(* Schneider Machine Expert - Basic project Questao3.3_FelipeV1_20241008, file version 2.9.0.0 *)
(* ProjectInformations: Name=Novo projeto *)

HARDWARE
  Cpu 0: TM221M16R/G
  EthernetConfiguration: NetworkName=M221, IpAllocationMode=FixedAddress, IpAddress=0.0.0.0, SubnetMask=0.0.0.0
  SerialLineConfiguration: Baud=Baud19200, Parity=ParityEven, DataBits=DataBits8, StopBits=StopBits1, PhysicalMedium=PhysicalMediumRs485, TransmissionMode=TransmissionModeModbusRtu, SlaveId=1, Addressing=SlaveAddressing
  MastTask: UsePeriodScanMode=false, PeriodScan=100
  FastTask: Period=255
  CpuBehavior: StartingMode=StartAsPreviousState, AutoSaveRamOnEeprom=true, WatchdogPeriod=250

SYMBOLS  (address, symbol, comment, settings)
  %M0       INIC_A_ATUA
  %M1       INIC_A_DESA
  %M2       INIC_B_ATUA
  %M3       INIC_B_DESA
  %M4       TEMP_A
  %M5       TEMP_B
  %M6       OK
  %M20      LIGA_PRENSA
  %TM0        "T1"  [Preset=3, Base=OneSecond]
  %TM1        [Preset=3, Base=OneSecond]
  %TM2        [Preset=3, Base=OneSecond]
  %I0.0     BOT_A_ATUA
  %I0.1     BOT_A_DESA
  %I0.2     BOT_B_ATUA
  %I0.3     BOT_B_DESA
  %Q0.0       "Contactor R"
  %Q0.1     PRENSA

POU Novo POU
  (* SectionNumber=0 *)

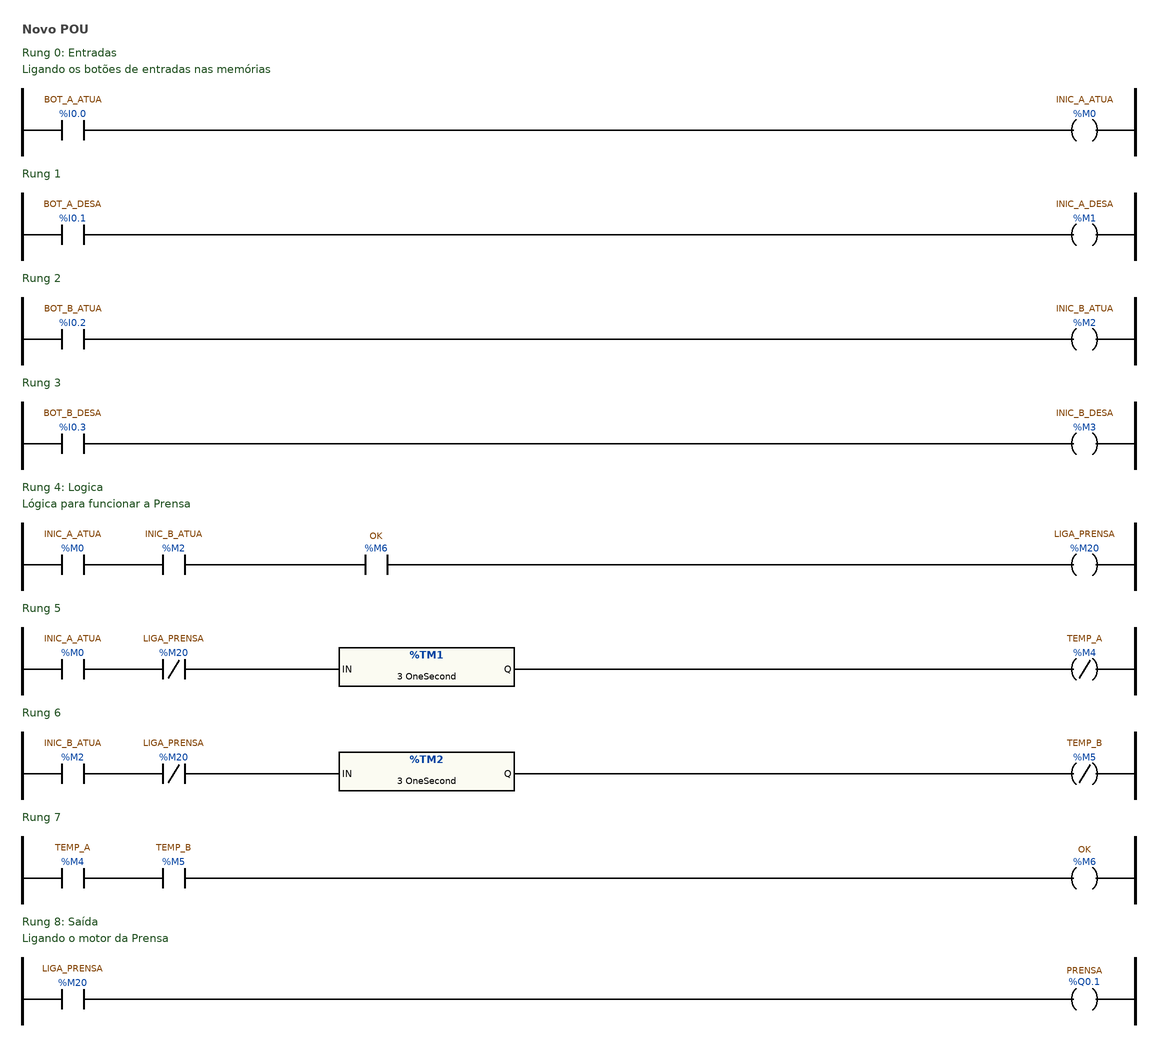

// Rung 0: Entradas
// Ligando os botões de entradas nas memórias
  LD %I0.0                (* BOT_A_ATUA *)
  ST %M0                  (* INIC_A_ATUA *)
  // as ST:
  //   INIC_A_ATUA := BOT_A_ATUA;

// Rung 1
  LD %I0.1                (* BOT_A_DESA *)
  ST %M1                  (* INIC_A_DESA *)
  // as ST:
  //   INIC_A_DESA := BOT_A_DESA;

// Rung 2
  LD %I0.2                (* BOT_B_ATUA *)
  ST %M2                  (* INIC_B_ATUA *)
  // as ST:
  //   INIC_B_ATUA := BOT_B_ATUA;

// Rung 3
  LD %I0.3                (* BOT_B_DESA *)
  ST %M3                  (* INIC_B_DESA *)
  // as ST:
  //   INIC_B_DESA := BOT_B_DESA;

// Rung 4: Logica
// Lógica para funcionar a Prensa
  LD %M0                  (* INIC_A_ATUA *)
  AND %M2                 (* INIC_B_ATUA *)
  AND %M6                 (* OK *)
  ST %M20                 (* LIGA_PRENSA *)
  // as ST:
  //   LIGA_PRENSA := INIC_A_ATUA AND INIC_B_ATUA AND OK;

// Rung 5
  BLK %TM1
  LD %M0                  (* INIC_A_ATUA *)
  ANDN %M20               (* LIGA_PRENSA *)
  IN
  OUT_BLK
  LD Q
  STN %M4                 (* TEMP_A *)
  END_BLK
  // as ST:
  //   %TM1(IN := INIC_A_ATUA AND NOT LIGA_PRENSA);
  //   TEMP_A := NOT %TM1.Q;

// Rung 6
  BLK %TM2
  LD %M2                  (* INIC_B_ATUA *)
  ANDN %M20               (* LIGA_PRENSA *)
  IN
  OUT_BLK
  LD Q
  STN %M5                 (* TEMP_B *)
  END_BLK
  // as ST:
  //   %TM2(IN := INIC_B_ATUA AND NOT LIGA_PRENSA);
  //   TEMP_B := NOT %TM2.Q;

// Rung 7
  LD %M4                  (* TEMP_A *)
  AND %M5                 (* TEMP_B *)
  ST %M6                  (* OK *)
  // as ST:
  //   OK := TEMP_A AND TEMP_B;

// Rung 8: Saída
// Ligando o motor da Prensa
  LD %M20                 (* LIGA_PRENSA *)
  ST %Q0.1                (* PRENSA *)
  // as ST:
  //   PRENSA := LIGA_PRENSA;
